FUNCTION alg_a_Hresetled : BOOL
VAR_INPUT
	state: STATE;
END_VAR

alg_a_Hresetled := FALSE;

END_FUNCTION

(* stored: Version 1.1.0.1, ProductVersion 3.1.4022.18
   POU alg_a_Hresetled: Id {aabf7912-d679-4ce7-b405-655f2ac7e013}, SpecialFunc None *)
